FUNCTION_BLOCK ExamplesImplementationWithDone EXTENDS TcoCore.TcoObject
VAR
    _inspectorsSignal : BOOL;
    _inspector        : TcoInspectors.TcoDigitalInspector(THIS^);
    _inspectorTask    : TcoCore.TcoTask(THIS^);
END_VAR

IF(_inspectorTask.Execute()) THEN	
	IF(_inspector.Inspect(_inspectorsSignal).Done) THEN
		IF(_inspector.Result = TcoInspectors.eInspectorResult.Failed) THEN
			_inspector.Messenger.Build().Append('I failed').As().AsInfo().Pin();
		ELSIF(_inspector.Result = TcoInspectors.eInspectorResult.Passed) THEN
			_inspector.Messenger.Build().Append('I passed').As().AsInfo().Pin();
		END_IF
	END_IF;		
END_IF;

END_FUNCTION_BLOCK

(* stored: Version 1.1.0.1, ProductVersion 3.1.4024.9
   POU ExamplesImplementationWithDone: Id {af9cd9f6-d43b-0818-0bd8-033f33b31536}, SpecialFunc None *)
